{attribute 'pack_mode' := '1'}
TYPE DUT_EpicsValueMetadata :
STRUCT

	fTimestamp : LREAL;
	nStatus : INT;
	nSeverity : INT;
	nDataType : BYTE;

END_STRUCT
END_TYPE

(* stored: Version 1.1.0.1, ProductVersion 3.1.4022.18
   DUT DUT_EpicsValueMetadata: Id {98f42ed6-e002-426b-a094-f3215801fad1} *)
